{attribute 'qualified_only'}
VAR_GLOBAL CONSTANT
	MAX_MOVERS			: INT 	:= 10;
	MAX_POSITIONS		: INT 	:= 10;
	MAX_POS_STATIONS	: INT 	:= 5;
	MAX_DEVICES 		: UDINT	:= 30;
	TRACK_LENGTH 		: LREAL := 3000;
END_VAR

(* stored: Version 1.1.0.1
   GVL SETTINGS: Id {d5b725cc-3025-4c4e-b484-c081e6746911}, ParameterList True *)
